PROGRAM MAIN
VAR
END_VAR

END_PROGRAM

(* stored: Version 1.1.0.1
   POU MAIN: Id {d5486261-b31a-4148-ac53-5edd2eed9164} *)
